{attribute 'qualified_only'}
VAR_GLOBAL
	
END_VAR

(* stored: Version 1.1.0.1, ProductVersion 3.1.4024.0
   GVL GVL: Id {c6edceb1-dcfd-40d2-850a-731dab31d70d} *)
